% RSLogix 500 project Inventory-Manager.RSS, saved by version 8.30.00.16 %
PROJECT "UNTITLED"    % processor: Bul.1763 MicroLogix 1100 Series B %

PROGRAM FILES
  LAD 2   10 rungs

DATA FILES
  O0 OUTPUT  4 elements
  I1 INPUT  6 elements
  S2 STATUS  66 elements
  B3 BINARY  1 elements
  T4 TIMER  1 elements
  C5 COUNTER  1 elements
  R6 CONTROL  1 elements
  N7 INTEGER  16 elements
  F8 FLOAT  1 elements
  ST9 SCAN  10 elements  % 9 %

LADDER 2
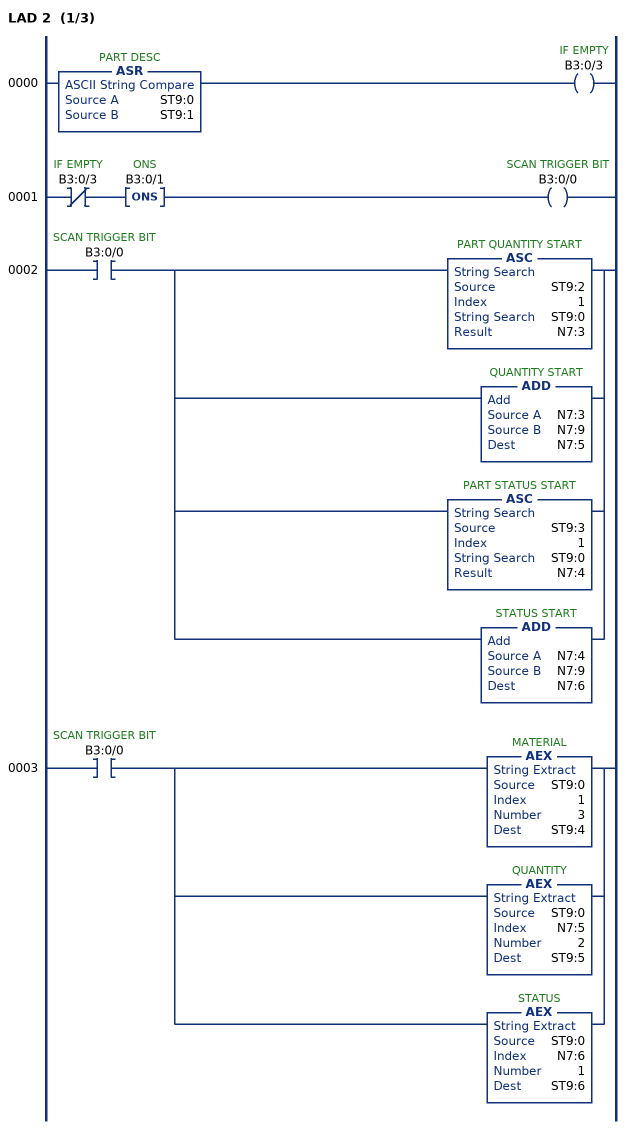
% Rung: 0 %
SOR ASR ST9:0 ST9:1 OTE B3:0/3 EOR
%   ST9:0  "PART DESC" %
%   ST9:1  "COMPARE IF EMPTY FOR SCAN" %
%   B3:0/3  "IF EMPTY" %
% Rung: 1 %
SOR XIO B3:0/3 ONS B3:0/1 OTE B3:0/0 EOR
%   B3:0/3  "IF EMPTY" %
%   B3:0/1  "ONS" %
%   B3:0/0  "SCAN TRIGGER BIT" %
% Rung: 2 %
SOR XIC B3:0/0 BST ASC ST9:2 1 ST9:0 N7:3 NXB ADD N7:3 N7:9 N7:5 NXB ASC ST9:3 1 ST9:0 N7:4 NXB ADD N7:4 N7:9 N7:6 BND EOR
%   B3:0/0  "SCAN TRIGGER BIT" %
%   ST9:2  "PART QUANTITY START" %
%   ST9:0  "PART DESC" %
%   N7:3  "QUANTITY START - 1" %
%   N7:9  "ADD 1" %
%   N7:5  "QUANTITY START" %
%   ST9:3  "PART STATUS START" %
%   N7:4  "STATUS START - 1" %
%   N7:6  "STATUS START" %
% Rung: 3 %
SOR XIC B3:0/0 BST AEX ST9:0 1 3 ST9:4 NXB AEX ST9:0 N7:5 2 ST9:5 NXB AEX ST9:0 N7:6 1 ST9:6 BND EOR
%   B3:0/0  "SCAN TRIGGER BIT" %
%   ST9:0  "PART DESC" %
%   ST9:4  "MATERIAL" %
%   N7:5  "QUANTITY START" %
%   ST9:5  "QUANTITY" %
%   N7:6  "STATUS START" %
%   ST9:6  "STATUS" %

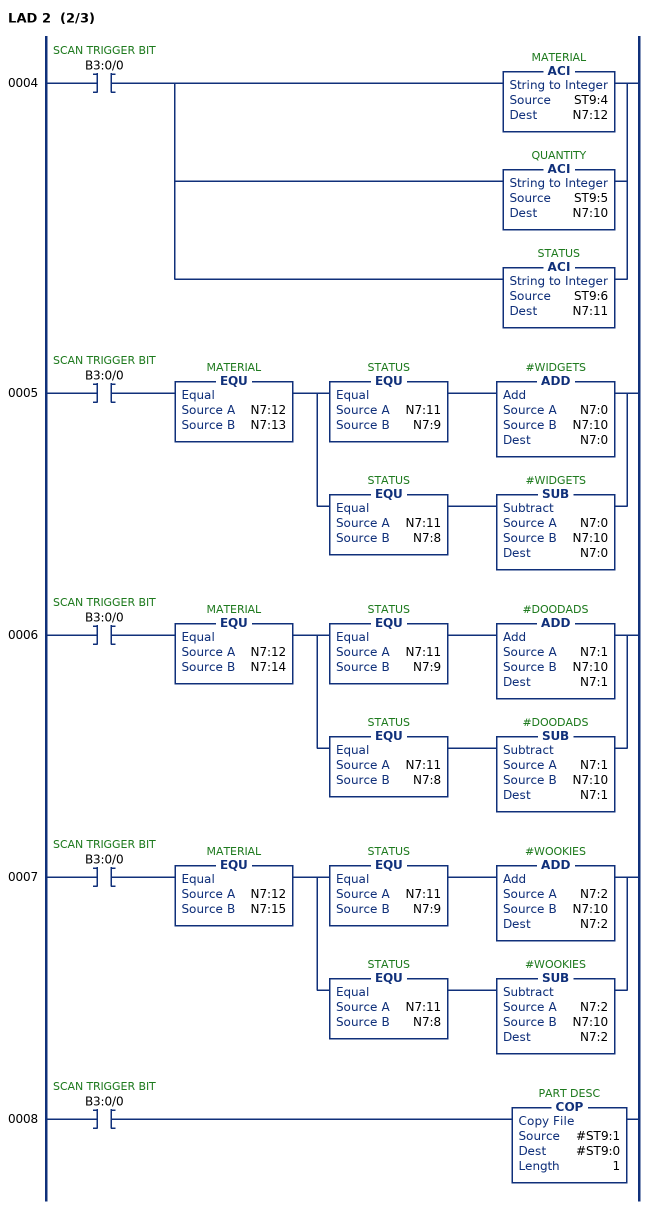
% Rung: 4 %
SOR XIC B3:0/0 BST ACI ST9:4 N7:12 NXB ACI ST9:5 N7:10 NXB ACI ST9:6 N7:11 BND EOR
%   B3:0/0  "SCAN TRIGGER BIT" %
%   ST9:4  "MATERIAL" %
%   N7:12  "MATERIAL" %
%   ST9:5  "QUANTITY" %
%   N7:10  "QUANTITY" %
%   ST9:6  "STATUS" %
%   N7:11  "STATUS" %
% Rung: 5 %
SOR XIC B3:0/0 EQU N7:12 N7:13 BST EQU N7:11 N7:9 ADD N7:0 N7:10 N7:0 NXB EQU N7:11 N7:8 SUB N7:0 N7:10 N7:0 BND EOR
%   B3:0/0  "SCAN TRIGGER BIT" %
%   N7:12  "MATERIAL" %
%   N7:13  "WIDGETS" %
%   N7:11  "STATUS" %
%   N7:9  "ADD 1" %
%   N7:0  "#WIDGETS" %
%   N7:10  "QUANTITY" %
%   N7:8  "COMPARE WITH ZERO FOR VALID SCAN" %
% Rung: 6 %
SOR XIC B3:0/0 EQU N7:12 N7:14 BST EQU N7:11 N7:9 ADD N7:1 N7:10 N7:1 NXB EQU N7:11 N7:8 SUB N7:1 N7:10 N7:1 BND EOR
%   B3:0/0  "SCAN TRIGGER BIT" %
%   N7:12  "MATERIAL" %
%   N7:14  "DOODADS" %
%   N7:11  "STATUS" %
%   N7:9  "ADD 1" %
%   N7:1  "#DOODADS" %
%   N7:10  "QUANTITY" %
%   N7:8  "COMPARE WITH ZERO FOR VALID SCAN" %
% Rung: 7 %
SOR XIC B3:0/0 EQU N7:12 N7:15 BST EQU N7:11 N7:9 ADD N7:2 N7:10 N7:2 NXB EQU N7:11 N7:8 SUB N7:2 N7:10 N7:2 BND EOR
%   B3:0/0  "SCAN TRIGGER BIT" %
%   N7:12  "MATERIAL" %
%   N7:15  "WOCKIES" %
%   N7:11  "STATUS" %
%   N7:9  "ADD 1" %
%   N7:2  "#WOOKIES" %
%   N7:10  "QUANTITY" %
%   N7:8  "COMPARE WITH ZERO FOR VALID SCAN" %
% Rung: 8 %
SOR XIC B3:0/0 COP #ST9:1 #ST9:0 1 EOR
%   B3:0/0  "SCAN TRIGGER BIT" %
%   ST9:1  "COMPARE IF EMPTY FOR SCAN" %
%   ST9:0  "PART DESC" %

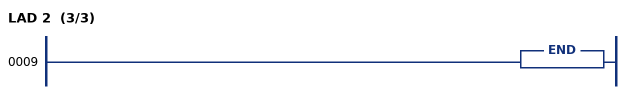
% Rung: 9 %
SOR END EOR

OTHER DOCUMENTED ADDRESSES
  B3:0/2  "SCAN ALWAYS ON"
  N7:0/3  "QUANTITY START"
  N7:0/4  "PART STATUS START"
  N7:0/5  N75  "QUANTITY START"
  N7:0/6  "STATUS START"
  N7:0/9  "ADD 1"
  N7:7  "COMPARE WITH ZERO"
  N7:10/0  "QUANTITY"
  N7:10/1  "STATUS"
  N7:10/2  "MATERIAL"
  N7:10/3  "WIDGETS"
  N7:10/4  "DOODADS"
  N7:10/5  "WOCKIES"
  ST9:9  "SCAN VARIABLE"

DATA TABLE (non-zero values as saved)
DATA B3
% B3:0 % 0X000C
DATA N7
% N7:0 % 1 15 30 4 7 5 8 0 0 1
% N7:10 % 19 0 123 123 456 789
DATA ST9
% ST9:2 % "-"
% ST9:3 % ":"
% ST9:4 % "123"
% ST9:5 % "19"
% ST9:6 % "0"
